(* CODESYS project SFC_RECOVERED_2024-07-03T18-49-14.project

Project tree, tasks and I/O mapping:
  Device : CODESYS Control Win V3, CODESYS, version 3.5.20.0
    application Application
      libraries: Standard, 3.5.18.0 (System)
      task MainTask (cyclic, interval t#20ms, priority 1) calls PLC_PRG
      task VISU_TASK (cyclic, interval 100 ms, priority 31) calls VisuElems.Visu_Prg
      visualisation Visualization
      program PLC_PRG [SFC]
  libraries: VisuSymbols, 4.5.0.0 (System)
  text list GlobalTextList
*)

// Device/Application/PLC_PRG
PROGRAM PLC_PRG
VAR
	StartPB:BOOL;
	PL:BOOL;
END_VAR

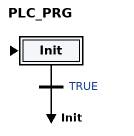
INITIAL_STEP Init:
END_STEP
TRANSITION FROM Init TO Init
    := TRUE;
END_TRANSITION

END_PROGRAM

// Device/Application/Visualization
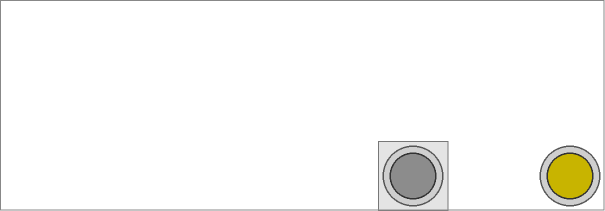
VISUALIZATION Visualization  // 605x211
    Lamp1 (535,141 70x70), style: Lamp-Lamp1-Yellow
    PushSwitch (378,141 70x70), behaviour: TOGGLE, style: Switch-PushSwitch-Gray
END_VISUALIZATION
